Yaskawa INFORM job: HOME.JBI

/JOB
//NAME HOME
//POS
///NPOS 1,0,0,0,0,0
///TOOL 0
///POSTYPE PULSE
///PULSE
C00000=-63952,-155163,126853,-105316,-81596,-126671
//INST
///DATE 2022/02/23 16:36
///ATTR SC,RW
///GROUP1 RB1
NOP
MOVJ C00000 VJ=65.00  //HOME
END
